//---------------------------------------------------------------------------------------------------------------
//
//  HAUD 2023.03.07
//
//  - XTS_TRANSPORT_LAYER
//
//  fb_Station
//  - handshake with extern control for mover transport through station
//
//---------------------------------------------------------------------------------------------------------------
// This SOFTWARE is provided as an Exemple by THE PROVIDER "as is" and "with all faults." THE PROVIDER makes no 
// representations or warranties of any kind concerning the safety, suitability, lack of viruses, inaccuracies, 
// typographical errors, or other harmful components of this SOFTWARE. There are inherent dangers in the use of 
// any software, and you are solely responsible for determining whether this SOFTWARE is compatible with your 
// equipment and other software installed on your equipment. You are also solely responsible for the protection 
// of your equipment and backup of your data, and THE PROVIDER will not be liable for any damages you may suffer 
// in connection with using, modifying, or distributing this SOFTWARE.
//---------------------------------------------------------------------------------------------------------------
FUNCTION_BLOCK fb_Station IMPLEMENTS I_XtsTransport_Station
VAR
  _nStationId                 : UINT;         // why is Gamora?

  _sState                     : STRING(255);  // additional output for Check()

  _eInitList                  : E_PROGRESS;   // linked list initialization progress

  _eFatalError                : E_STATION_STATE;

  // pointer to all stations
  _stCtrl                     : REFERENCE TO ARRAY[1..MAX_STATION]  OF ST_STATION_CTRL;
  _stState                    : REFERENCE TO ARRAY[1..MAX_STATION]  OF ST_STATION_STATE;

  // local copy of command
  _eCmd,
  _eCmdOld                    : E_STATION_CTRL;

  _ItfStation                 : REFERENCE TO ARRAY[1..MAX_STATION]  OF I_Station_LinkedList;  // access to all stations lists
  _ItfMover                   : REFERENCE TO ARRAY[1..MAX_MOVER]    OF I_XtsTransport_Mover;  // access to mover methods

  // station related data
  _rMoverOffset               : REFERENCE TO ARRAY[1..MAX_STATION]  OF T_NEST_OFFSET;         // static offsets for station
  _stParameter                : REFERENCE TO ARRAY[1..MAX_STATION]  OF ST_STATION_PARAMETER;  // station parameter (where, how fast, how many stops)

  // mover axis ref for info
  _Mover                      : REFERENCE TO ARRAY[1..MAX_MOVER]    OF AXIS_REF;              // read from AXIS_REF

  // linked list result struct
  _stListEnter,
  _stListTarget,
  _stListDelete               : ST_STATION_LIST_RESULT;   // struct with result and ticket data

  _stMoverDataSend,
  _stMoverData                : ST_STATION_MOVER_DATA;    // mover ticket data

  _stInfeed,
  _stOutfeed                  : ST_MOVE_DATA;             // position and dynamic constraints of movement

  // work vars
  _Result                     : E_PROGRESS;
  _eStateProgress             : E_PROGRESS;

  _nNest,
  _nMoverDetected,
  _ix                         : UINT;

  _rModActPosFetch            : LREAL;
  _stMsg                      : ST_Message;
  _eMessageLevel              : E_MessageType;
END_VAR

METHOD PRIVATE Check : BOOL
VAR_INPUT
END_VAR
IF NOT (_nStationId > 0) OR
       (_nStationId > MAX_STATION)
THEN
  _sState                     := 'invalid nStationId';
  RETURN;
END_IF

IF NOT __ISVALIDREF(_stCtrl)
THEN
  _sState                     := '_stCtrl: missing pointer';
  RETURN;
END_IF

IF NOT __ISVALIDREF(_stState)
THEN
  _sState                     := '_stState: missing pointer';
  RETURN;
END_IF

IF NOT __ISVALIDREF(_ItfStation)
THEN
  _sState                     := '_ItfStation: missing interface';
  RETURN;
END_IF

IF NOT __ISVALIDREF(_ItfMover)
THEN
  _sState                     := '_ItfMover: missing interface';
  RETURN;
END_IF

IF NOT __ISVALIDREF(_rMoverOffset)
THEN
  _sState                     := '_rMoverOffset: missing pointer';
  RETURN;
END_IF

IF NOT __ISVALIDREF(_stParameter)
THEN
  _sState                     := '_stParameter: missing pointer';
  RETURN;
END_IF

IF NOT __ISVALIDREF(_Mover)
THEN
  _sState                     := '_Mover: missing pointer';
  RETURN;
END_IF


_sState                       := 'CHECK_DONE';
Check                         := TRUE;
END_METHOD

PROPERTY Ctrl : reference to ARRAY[1..MAX_STATION] OF ST_STATION_CTRL
SET
_stCtrl ref= Ctrl;
END_SET
END_PROPERTY

METHOD Cycle
//-----------------------------------------------------------------------------
//-----------------------------------------------------------------------------
// check pointer and interface
//-----------------------------------------------------------------------------
IF NOT Check() THEN RETURN; END_IF
//-----------------------------------------------------------------------------
//-----------------------------------------------------------------------------
// set message device ID
//-----------------------------------------------------------------------------
_stMsg.eDevice                        := e_Device.XtsStation + _nStationId;
//-----------------------------------------------------------------------------
//-----------------------------------------------------------------------------
// log command change
//-----------------------------------------------------------------------------
_eCmd                                 := _stCtrl[_nStationId].eCmd;
IF (_eCmd <> _eCmdOld)
THEN
  _eCmdOld                            := _eCmd;

  _stMsg.eType                        := E_MessageType.eMessageInfo;
  _stMsg.eSubdevice                   := StationControl;
  _stMsg.iErrorNumber                 := 0;
  _stMsg.sText                        := TO_STRING(_eCmd);

  IF (_eMessageLevel > E_MessageType.eMessageWarning)
  THEN
    f_MessageSet(_stMsg);
  END_IF
END_IF
//-----------------------------------------------------------------------------
//-----------------------------------------------------------------------------
// clear station on demand
//-----------------------------------------------------------------------------
CASE _stCtrl[_nStationId].eCmd
OF
  E_STATION_CTRL.STATION_INIT:        // commanded init from cyclic interface
    _eInitList                        := Init();
    _stState[_nStationId].rMoverModPos:= 0.0;
    _stState[_nStationId].nQueue      := TO_USINT(_ItfStation[_nStationId].Count);
    RETURN;
END_CASE
//-----------------------------------------------------------------------------
//-----------------------------------------------------------------------------
// station startup and init states
//-----------------------------------------------------------------------------
CASE _stState[_nStationId].eState
OF
  E_STATION_STATE.STATION_NO_INIT:    // startup state in first PLC cycle, init linked list required
    _eInitList                        := Init();

  E_STATION_STATE.STATION_INIT:       // switch state as reserve for anything you might add here
    _stState[_nStationId].eState      := E_STATION_STATE.STATION_DISABLE;
END_CASE
//-----------------------------------------------------------------------------
//-----------------------------------------------------------------------------
//  station disabled after init 
//  wait for command to enable
//  return state after a mover has left station
//  fall back state before entry was allowed and you decided to disable
//-----------------------------------------------------------------------------
CASE _stState[_nStationId].eState
OF
  E_STATION_STATE.STATION_DISABLE:
    IF (_stCtrl[_nStationId].eCmd = E_STATION_CTRL.STATION_ENABLE)
    THEN
      _stState[_nStationId].eState    := E_STATION_STATE.STATION_ENABLE;
    END_IF


  E_STATION_STATE.STATION_ENABLE:     // enable state is detectable on the interface for one cycle only
                                      // double check commanded enable and clear work vars
    IF (_stCtrl[_nStationId].eCmd = E_STATION_CTRL.STATION_DISABLE)
    THEN
      _stState[_nStationId].eState    := E_STATION_STATE.STATION_DISABLE;
    ELSE
      memset(ADR(_stListEnter),    0, SIZEOF(_stListEnter));

      _eStateProgress                 := E_PROGRESS.PROGRESS_INIT;  // substate for procedures within one state
      _stState[_nStationId].eState    := E_STATION_STATE.STATION_DETECT_MOVER;  // switch to mover detection

      IF (_eMessageLevel = E_MessageType.eMessageVerbose)
      THEN
        _stMsg.eType                  := _eMessageLevel;
        LogState(_stMsg.eType);
      END_IF
    END_IF
END_CASE
//-----------------------------------------------------------------------------
//-----------------------------------------------------------------------------
//  detection state
//   - wait until mover data is entered into list
//
//  check for disable command; fall back to disabled state
//  check linked list for new entry; proceed to request infeed of mover
//-----------------------------------------------------------------------------
CASE _stState[_nStationId].eState
OF
  E_STATION_STATE.STATION_DETECT_MOVER:// wait state for mover detection
    CASE _eStateProgress
    OF
      E_PROGRESS.PROGRESS_INIT:
        IF (_stCtrl[_nStationId].eCmd = E_STATION_CTRL.STATION_DISABLE) // check for commanded disable
        THEN
          IF (_eMessageLevel = E_MessageType.eMessageVerbose)
          THEN
            _stMsg.eType              := E_MessageType.eMessageVerbose;
            _stMsg.eSubdevice         := Stationstate;
            _stMsg.iErrorNumber       := _stState[_nStationId].nMoverId;
            _stMsg.sText              := concat(TO_STRING(_stState[_nStationId].eState), ': ');
            _stMsg.sText              := concat(_stMsg.sText, TO_STRING(E_STATION_STATE.STATION_DISABLE));
            f_MessageSet(_stMsg);
          END_IF
          _stState[_nStationId].eState      := E_STATION_STATE.STATION_DISABLE; // go back and wait, no matter the queue

        ELSIF (_ItfStation[_nStationId].Count > 0)
        THEN
          // someone entered something in my list
          _stListEnter                := _ItfStation[_nStationId].GetHead();
          _eStateProgress             := E_PROGRESS.PROGRESS_BUSY;  // go check list result data

          IF (_eMessageLevel > E_MessageType.eMessageWarning)
          THEN
            _stMsg.eType              := E_MessageType.eMessageInfo;
            _stMsg.eSubdevice         := Stationstate;
            _stMsg.iErrorNumber       := _stState[_nStationId].nMoverId;
            _stMsg.sText              := concat(TO_STRING(_stState[_nStationId].eState), ': ');
            _stMsg.sText              := concat(_stMsg.sText, TO_STRING(_eStateProgress));
            f_MessageSet(_stMsg);
          END_IF
        END_IF
    END_CASE
    CASE _eStateProgress
    OF
      E_PROGRESS.PROGRESS_BUSY:
        IF (_stListEnter.wState = 0)  // GetHead() without error
        THEN
          _stMsg.eType                := E_MessageType.eMessageVerbose;
          _stMsg.eSubdevice           := e_Subdevice.StationGetHead;
          _stMsg.iErrorNumber         := _stListEnter.stData.nMoverId;
          _stMsg.sText                := '';
          IF (_eMessageLevel = E_MessageType.eMessageVerbose)
          THEN
            f_MessageSet(_stMsg);
          END_IF

          // list is giving head as result
          _stMoverData                := _stListEnter.stData; // copy ticket from list result
          _eStateProgress             := E_PROGRESS.PROGRESS_PREPARE; // go check plausibility of ticket

          IF (_eMessageLevel = E_MessageType.eMessageVerbose)
          THEN
            _stMsg.eType              := E_MessageType.eMessageVerbose;
            _stMsg.eSubdevice         := Stationstate;
            _stMsg.iErrorNumber       := _stState[_nStationId].nMoverId;
            _stMsg.sText              := concat(TO_STRING(_stState[_nStationId].eState), ': ');
            _stMsg.sText              := concat(_stMsg.sText, TO_STRING(_eStateProgress));
            f_MessageSet(_stMsg);
          END_IF
        ELSE
          // the thing that must not be: GetHead() with error
          _stState[_nStationId].eState      := E_STATION_STATE.STATION_ERROR_LIST_GET_HEAD_FAULT; // fatal error

          _stMsg.eType                      := E_MessageType.eMessageError;
          LogState(_stMsg.eType);
        END_IF
    END_CASE
    CASE _eStateProgress
    OF
      E_PROGRESS.PROGRESS_PREPARE:    // check ticket (list entry)
        // check target assignement
        IF NOT (_stMoverData.nTargetStation = _nStationId)
        THEN
          // for whom the mover calls
          // wrong address, right mover?
          _stState[_nStationId].eState      := E_STATION_STATE.STATION_ERROR_LIST_STATION_ID_WRONG; // ctrl has to fix this, go tell ctrl

          _stMsg.eType                      := E_MessageType.eMessageWarning;
          LogState(_stMsg.eType);
        ELSE
          // it's a me
          _nMoverDetected                   := _stMoverData.nMoverId;

          IF (_nMoverDetected < 1) OR
             (_nMoverDetected > MAX_MOVER)
          THEN
            // out of range the mover must not be
            _stState[_nStationId].eState    := E_STATION_STATE.STATION_ERROR_LIST_MOVER_ID_INVALID; // fatal error

            _stMsg.eType                    := E_MessageType.eMessageError;
            LogState(_stMsg.eType);
          ELSE
            memset(ADR(_stListDelete),   0, SIZEOF(_stListDelete)); // clear work var
            _eStateProgress                 := E_PROGRESS.PROGRESS_INIT; // clear progress for next station state

            // prepare station state for new mover
            _stState[_nStationId].nMoverId  := TO_USINT(_nMoverDetected); // who is waiting to enter
            _stState[_nStationId].nMask     := _stMoverData.nMask;        // how many stops have to be made
            _stState[_nStationId].eState    := E_STATION_STATE.STATION_MOVER_ENTER; // go ask for permission to enter

            IF (_eMessageLevel > E_MessageType.eMessageWarning)
            THEN
              _stMsg.eType            := E_MessageType.eMessageInfo;
              _stMsg.eSubdevice       := Stationstate;
              _stMsg.iErrorNumber     := _stState[_nStationId].nMoverId;
              _stMsg.sText            := concat(TO_STRING(_stState[_nStationId].eState), ': ');
              _stMsg.sText            := concat(_stMsg.sText, TO_STRING(_eStateProgress));
              f_MessageSet(_stMsg);
            END_IF
          END_IF
        END_IF
    END_CASE
END_CASE
//-----------------------------------------------------------------------------
//-----------------------------------------------------------------------------
// enter into station state
//  last check for disable command; fall back to disabled state
//  check for command to enter; prepare moverment, start movement
//  check for command to skip; prepare movement, switch to outfeed state
//-----------------------------------------------------------------------------
CASE _stState[_nStationId].eState
OF
  E_STATION_STATE.STATION_MOVER_ENTER:          // requesting permission for mover to enter station
    CASE _eStateProgress
    OF
      E_PROGRESS.PROGRESS_INIT:

        CASE _stCtrl[_nStationId].eCmd
        OF
          E_STATION_CTRL.STATION_DISABLE:       // control decided to disable, mover will wait
            _stState[_nStationId].eState    := E_STATION_STATE.STATION_DISABLE;

            IF (_eMessageLevel = E_MessageType.eMessageVerbose)
            THEN
              _stMsg.eType                  := _eMessageLevel;
              LogState(_stMsg.eType);
            END_IF

          E_STATION_CTRL.STATION_MOVER_ENTER:   // control decided to let mover enter
            _nNest                    := 1;     // default nest/PosStop[1]
            _eStateProgress           := E_PROGRESS.PROGRESS_BUSY;

            IF (_eMessageLevel = E_MessageType.eMessageVerbose)
            THEN
              _stMsg.eType            := E_MessageType.eMessageVerbose;
              _stMsg.eSubdevice       := Stationstate;
              _stMsg.iErrorNumber     := _stState[_nStationId].nMoverId;
              _stMsg.sText            := concat(TO_STRING(_stState[_nStationId].eState), ': ');
              _stMsg.sText            := concat(_stMsg.sText, TO_STRING(_eStateProgress));
              f_MessageSet(_stMsg);
            END_IF

            FOR _ix := 1 TO _stParameter[_nStationId].nConfiguredStopCount
            DO
              IF GetBitWord(_stMoverData.nMask, _ix-1)
              THEN
                _nNest                := _ix;
                EXIT;
              END_IF
            END_FOR

          E_STATION_CTRL.STATION_MOVER_SEND:    // control decided to send mover away
            _stOutfeed.rDistance          := _stParameter[_nStationId].rReleaseDistance;
            _stState[_nStationId].eState  := E_STATION_STATE.STATION_MOVER_OUT;

            IF (_eMessageLevel = E_MessageType.eMessageVerbose)
            THEN
              _stMsg.eType                := _eMessageLevel;
              LogState(_stMsg.eType);
            END_IF
        END_CASE
    END_CASE
    CASE _eStateProgress
    OF
      E_PROGRESS.PROGRESS_BUSY:
        MoveData();                   // prepare movement into station

        // check if infeed movement has to cross modulo turn
        _rModActPosFetch              := _Mover[_stMoverData.nMoverId].NcToPlc.ModuloActPos;

        IF (_rModActPosFetch > _stInfeed.rPos + _stParameter[_nStationId].rReleaseDistance)
        THEN
          _stInfeed.rPos              := _stInfeed.rPos + TO_REAL(_ItfMover[_stMoverData.nMoverId].RailLength);
        END_IF

        _stState[_nStationId].eState  := E_STATION_STATE.STATION_MOVER_IN_TARGET;

        IF (_eMessageLevel = E_MessageType.eMessageVerbose)
        THEN
          _stMsg.eType                := _eMessageLevel;
          LogState(_stMsg.eType);
        END_IF
    END_CASE
END_CASE
//-----------------------------------------------------------------------------
//-----------------------------------------------------------------------------
// move into station state
//  wait for movement to be done; mover in position and standstill
//    switch state to process handshake
//-----------------------------------------------------------------------------
CASE _stState[_nStationId].eState
OF
  E_STATION_STATE.STATION_MOVER_IN_TARGET:
    _ItfMover[_stMoverData.nMoverId].MessageLevel := _eMessageLevel;

    _Result := _ItfMover[_stState[_nStationId].nMoverId].MoveToPosCa(TRUE, _stInfeed);

    IF (_Result = E_PROGRESS.PROGRESS_DONE)
    THEN
      // mother! has arrived
      _ItfMover[_stState[_nStationId].nMoverId].MoveToPosCa(FALSE, _stInfeed);
      _stState[_nStationId].eState    := E_STATION_STATE.STATION_PROCESS_START;

      IF (_eMessageLevel > E_MessageType.eMessageWarning)
      THEN
        _stMsg.eType                  := E_MessageType.eMessageInfo;
        LogState(_stMsg.eType);
      END_IF
    ELSE
      IF (_Result = E_PROGRESS.PROGRESS_ERROR)
      THEN
        _ItfMover[_stState[_nStationId].nMoverId].MoveToPosCa(FALSE, _stInfeed);
        _stState[_nStationId].eState  := E_STATION_STATE.STATION_ERROR_INFEED_ERROR; // ctrl has to fix this, go tell ctrl

        _stMsg.eType                  := E_MessageType.eMessageError;
        LogState(_stMsg.eType);
      END_IF 
    END_IF
END_CASE
//-----------------------------------------------------------------------------
//-----------------------------------------------------------------------------
// process handshake state
//  clear bit in mask
//-----------------------------------------------------------------------------
CASE _stState[_nStationId].eState
OF
  E_STATION_STATE.STATION_PROCESS_START:
    IF (_stCtrl[_nStationId].eCmd = E_STATION_CTRL.STATION_PROCESS_START) OR  // double handshake, your choice
       (_stCtrl[_nStationId].eCmd = E_STATION_CTRL.STATION_PROCESS_DONE)      // single handshake, your choice
    THEN
      // clear bit in mask when started/done
      _stState[_nStationId].nMask     := TO_USINT(DelBitWord(TO_WORD(_stState[_nStationId].nMask), _nNest-1));
      _stState[_nStationId].eState    := E_STATION_STATE.STATION_PROCESS_DONE;

      IF (_eMessageLevel = E_MessageType.eMessageVerbose)
      THEN
        _stMsg.eType                  := _eMessageLevel;
        LogState(_stMsg.eType);
      END_IF
    END_IF
END_CASE
//-----------------------------------------------------------------------------
//-----------------------------------------------------------------------------
CASE _stState[_nStationId].eState
OF
  E_STATION_STATE.STATION_PROCESS_DONE:
    IF (_stCtrl[_nStationId].eCmd = E_STATION_CTRL.STATION_PROCESS_DONE)
    THEN
      _stState[_nStationId].eState    := E_STATION_STATE.STATION_CHECK;
    END_IF
END_CASE
//-----------------------------------------------------------------------------
//-----------------------------------------------------------------------------
// check state if the mover has to move to another nest or must leave station
//-----------------------------------------------------------------------------
CASE _stState[_nStationId].eState
OF
  E_STATION_STATE.STATION_CHECK:
    IF (_stState[_nStationId].nMask = 0)
    THEN
      // mover has to leave
      _stState[_nStationId].eState    := E_STATION_STATE.STATION_MOVER_OUT;

      IF (_eMessageLevel = E_MessageType.eMessageVerbose)
      THEN
        _stMsg.eType                  := _eMessageLevel;
        LogState(_stMsg.eType);
      END_IF
    ELSE
      // _stState[_nStationId].nMask <> 0
      FOR _ix := 1 TO MAX_STATION_NEST
      DO
        IF NOT (_ix > _stParameter[_nStationId].nConfiguredStopCount)
        THEN
          IF GetBitWord(_stState[_nStationId].nMask, _ix-1)
          THEN
            // more work to do
            _stState[_nStationId].eState  := E_STATION_STATE.STATION_CHECK_NEST;
            _nNest                        := _ix; // index to move to

            IF (_eMessageLevel = E_MessageType.eMessageVerbose)
            THEN
              _stMsg.eType                := _eMessageLevel;
              LogState(_stMsg.eType);
            END_IF
            EXIT;
          END_IF
        ELSE
          IF GetBitWord(_stState[_nStationId].nMask, _ix-1)
          THEN
            // not configured, not worked
            _stMsg.eType              := E_MessageType.eMessageWarning;
            _stMsg.eSubdevice         := Stationstate;
            _stMsg.iErrorNumber       := _ix;
            _stMsg.sText              := concat(TO_STRING(_stState[_nStationId].eState), ': ');
            _stMsg.sText              := concat(_stMsg.sText, Tc2_Utilities.BYTE_TO_BINSTR(_stState[_nStationId].nMask, TO_INT(MAX_STATION_NEST)));
            IF (_eMessageLevel > E_MessageType.eMessageError)
            THEN
              f_MessageSet(_stMsg);
            END_IF

            _stState[_nStationId].nMask := TO_USINT(DelBitWord(TO_WORD(_stState[_nStationId].nMask), _ix-1));
          END_IF
        END_IF
      END_FOR
    END_IF
END_CASE
//-----------------------------------------------------------------------------
//-----------------------------------------------------------------------------
// wait state before movement to next nest has to be started
//-----------------------------------------------------------------------------
CASE _stState[_nStationId].eState
OF
  E_STATION_STATE.STATION_CHECK_NEST:
    MoveData();

    IF (_stCtrl[_nStationId].eCmd = E_STATION_CTRL.STATION_MOVER_ENTER)
    THEN
      _stState[_nStationId].eState    := E_STATION_STATE.STATION_MOVER_IN_TARGET;
  
      IF (_eMessageLevel = E_MessageType.eMessageVerbose)
      THEN
        _stMsg.eType                  := _eMessageLevel;
        LogState(_stMsg.eType);
      END_IF
    END_IF
END_CASE
//-----------------------------------------------------------------------------
//-----------------------------------------------------------------------------
// wait state for outfeed of mover
//  check ctrl data, target must be plausible, nTargetStation is what you have to set
//-----------------------------------------------------------------------------
CASE _stState[_nStationId].eState
OF
  E_STATION_STATE.STATION_MOVER_OUT:
    IF (_stCtrl[_nStationId].eCmd = E_STATION_CTRL.STATION_MOVER_OUT)
    THEN
      IF (_stCtrl[_nStationId].nTargetStation < 1) OR  
         (_stCtrl[_nStationId].nTargetStation > MAX_STATION)
      THEN
        _stState[_nStationId].eState  := E_STATION_STATE.STATION_ERROR_OUTFEED_TARGET_INVALID; // ctrl has to fix this, go tell ctrl

        _stMsg.eType                  := E_MessageType.eMessageError;
        LogState(_stMsg.eType);
      ELSE
        _stListDelete                 := _ItfStation[_nStationId].RemoveHeadValue(); // delete mover data in stations linked list


        IF (_stListDelete.wState <> 0)
        THEN
        // deleting mover in list was NOT successful
          _stState[_nStationId].eState:= E_STATION_STATE.STATION_ERROR_LIST_REMOVE_HEAD_FAULT; // fatal error

          _stMsg.eType                := E_MessageType.eMessageError;
          LogState(_stMsg.eType);

        ELSE
        // mover data successfully deleted
          _stMsg.eType                := E_MessageType.eMessageVerbose;
          _stMsg.eSubdevice           := e_Subdevice.StationRemoveHeadValue;
          _stMsg.iErrorNumber         := _stState[_nStationId].nMoverId;
          _stMsg.sText                := '';
          IF (_eMessageLevel = E_MessageType.eMessageVerbose)
          THEN
            f_MessageSet(_stMsg);
          END_IF

          memset(ADR(_stListTarget),   0, SIZEOF(_stListTarget)); // clear debug var

          // prepare movement and switch state to start movement
          MoverOut();
          _stState[_nStationId].eState  := E_STATION_STATE.STATION_MOVER_RELEASE;

          IF (_eMessageLevel > E_MessageType.eMessageWarning)
          THEN
            _stMsg.eType                := E_MessageType.eMessageInfo;
            LogState(_stMsg.eType);
          END_IF
        END_IF
      END_IF
    END_IF
END_CASE
//-----------------------------------------------------------------------------
//-----------------------------------------------------------------------------
// ckeck if mover has left the station
//  enter mover data into list of target station
//-----------------------------------------------------------------------------
CASE _stState[_nStationId].eState
OF
  E_STATION_STATE.STATION_MOVER_RELEASE:
    _ItfMover[_stMoverData.nMoverId].MessageLevel := _eMessageLevel;

    _Result                           := _ItfMover[_stMoverDataSend.nMoverId].SendToModuloPosCa(TRUE, _stOutfeed);

    IF (_Result = E_PROGRESS.PROGRESS_DONE)
    THEN
      // add entry in target station list
      _stListTarget                   := _ItfStation[_stMoverDataSend.nTargetStation].AddTailValue(_stMoverDataSend);

      IF (_stListTarget.wState <> 0)
      THEN
      // adding mover in target list was NOT successful
        _stState[_nStationId].eState  := E_STATION_STATE.STATION_ERROR_LIST_ADD_TAIL_FAULT; // fatal error
        _stMsg.eType                  := E_MessageType.eMessageError;
        LogState(_stMsg.eType);

      ELSE
      // mover data successfully added to target station list
        IF (_eMessageLevel > E_MessageType.eMessageWarning)
        THEN
          _stMsg.eType                := E_MessageType.eMessageInfo;
          _stMsg.eSubdevice           := e_Subdevice.StationAddTail;
          _stMsg.iErrorNumber         := _stState[_nStationId].nMoverId;
          _stMsg.sText                := concat('TargetStation: ', TO_STRING(_stListTarget.stData.nTargetStation));
          f_MessageSet(_stMsg);
        END_IF

        _stState[_nStationId].eState  := E_STATION_STATE.STATION_MOVER_GONE; // go tell ctrl that station is empty

        IF (_eMessageLevel = E_MessageType.eMessageVerbose)
        THEN
          _stMsg.eType                := _eMessageLevel;
          LogState(_stMsg.eType);
        END_IF
      END_IF
    ELSIF (_Result = E_PROGRESS.PROGRESS_ERROR)
    THEN
      _stState[_nStationId].eState    := E_STATION_STATE.STATION_ERROR_OUTFEED_ERROR; // ctrl has to fix this, go tell ctrl
      _stMsg.eType                    := E_MessageType.eMessageError;
      LogState(_stMsg.eType);
    END_IF
END_CASE
//-----------------------------------------------------------------------------
//-----------------------------------------------------------------------------
// check handshake for empty station
//  switch back station state for new mover to be able to enter
//-----------------------------------------------------------------------------
CASE _stState[_nStationId].eState
OF
  E_STATION_STATE.STATION_MOVER_GONE:
    _ItfMover[_stMoverDataSend.nMoverId].SendToModuloPosCa(FALSE, _stOutfeed);

    memset(ADR(_stMoverData),  0, SIZEOF(_stMoverData));

    _stState[_nStationId].nMask       := 0;
    _stState[_nStationId].nMoverId    := 0;

    IF (_stCtrl[_nStationId].eCmd = E_STATION_CTRL.STATION_MOVER_GONE)
    THEN
      _stState[_nStationId].eState    := E_STATION_STATE.STATION_DISABLE;

      IF (_eMessageLevel = E_MessageType.eMessageVerbose)
      THEN
        _stMsg.eType                  := _eMessageLevel;
        LogState(_stMsg.eType);
      END_IF
    END_IF
END_CASE
//-----------------------------------------------------------------------------
//-----------------------------------------------------------------------------
_sState                               := TO_STRING(_stState[_nStationId].eState);
//-----------------------------------------------------------------------------
//-----------------------------------------------------------------------------
// Error handling
//-----------------------------------------------------------------------------
CASE _stState[_nStationId].eState
OF
  //---------------------------------------------------------------------------
  //---------------------------------------------------------------------------
  E_STATION_STATE.STATION_ERROR_LIST_STATION_ID_WRONG:
    IF (_stCtrl[_nStationId].eCmd = E_STATION_CTRL.STATION_MOVER_OUT)
    THEN
      _nMoverDetected                 := _stMoverData.nMoverId;

      IF (_nMoverDetected < 1) OR
         (_nMoverDetected > MAX_MOVER)
      THEN
        // this MUST NOT happen
        _stState[_nStationId].eState  := E_STATION_STATE.STATION_ERROR_LIST_MOVER_ID_INVALID; // fatal error
        _stMsg.eType                  := E_MessageType.eMessageError;
        LogState(_stMsg.eType);

      ELSE
        // not for station; send mover out
        _stState[_nStationId].eState  := E_STATION_STATE.STATION_MOVER_OUT;

        IF (_eMessageLevel > E_MessageType.eMessageError)
        THEN
          _stMsg.eType                := E_MessageType.eMessageInfo;
          LogState(_stMsg.eType);
        END_IF
      END_IF

    ELSIF (_stCtrl[_nStationId].eCmd = E_STATION_CTRL.STATION_MOVER_ENTER)
    THEN
      // override wrong TargetStationId in List; start infeed of mover

      _nMoverDetected                 := _stMoverData.nMoverId;

      IF (_nMoverDetected < 1) OR
         (_nMoverDetected > MAX_MOVER)
      THEN
        // this MUST NOT happen
        _stState[_nStationId].eState  := E_STATION_STATE.STATION_ERROR_LIST_MOVER_ID_INVALID; // fatal error

        _stMsg.eType                  := E_MessageType.eMessageError;
        LogState(_stMsg.eType);

      ELSE
        _eStateProgress               := E_PROGRESS.PROGRESS_INIT;
        _stState[_nStationId].nMoverId:= TO_USINT(_nMoverDetected);
        _stState[_nStationId].nMask   := _stMoverData.nMask;
        _stState[_nStationId].eState  := E_STATION_STATE.STATION_MOVER_ENTER;

        IF (_eMessageLevel > E_MessageType.eMessageError)
        THEN
          _stMsg.eType                := E_MessageType.eMessageInfo;
          LogState(_stMsg.eType);
        END_IF
      END_IF
    END_IF

  //---------------------------------------------------------------------------
  //---------------------------------------------------------------------------
  E_STATION_STATE.STATION_ERROR_OUTFEED_TARGET_INVALID:
    // wait here until valid target is detected
    IF NOT (_stCtrl[_nStationId].nTargetStation < 1) AND  
       NOT (_stCtrl[_nStationId].nTargetStation > MAX_STATION)
    THEN
      _stState[_nStationId].eState    := E_STATION_STATE.STATION_MOVER_OUT;

      IF (_eMessageLevel > E_MessageType.eMessageError)
      THEN
        _stMsg.eType                  := E_MessageType.eMessageInfo;
        LogState(_stMsg.eType);
      END_IF
    END_IF

  //---------------------------------------------------------------------------
  //---------------------------------------------------------------------------
  E_STATION_STATE.STATION_ERROR_INFEED_ERROR:   // must be fixed by extern by using cyclic mover control
    IF (_stCtrl[_nStationId].eCmd = E_STATION_CTRL.STATION_MOVER_ENTER_RETRY)
    THEN
      _stState[_nStationId].eState    := E_STATION_STATE.STATION_DETECT_MOVER;   // return to start and wait

      IF (_eMessageLevel > E_MessageType.eMessageError)
      THEN
        _stMsg.eType                  := E_MessageType.eMessageInfo;
        LogState(_stMsg.eType);
      END_IF
    END_IF


  //---------------------------------------------------------------------------
  //---------------------------------------------------------------------------
  E_STATION_STATE.STATION_ERROR_OUTFEED_ERROR:  // must be fixed by extern by using cyclic mover control
    IF (_stCtrl[_nStationId].eCmd = E_STATION_CTRL.STATION_MOVER_OUT_RETRY)
    THEN
      _stState[_nStationId].eState    := E_STATION_STATE.STATION_MOVER_OUT; // return to send out and wait

      IF (_eMessageLevel > E_MessageType.eMessageError)
      THEN
        _stMsg.eType                  := E_MessageType.eMessageInfo;
        LogState(_stMsg.eType);
      END_IF

    ELSIF (_stCtrl[_nStationId].eCmd = E_STATION_CTRL.STATION_MOVER_GONE)
    THEN
      MoverOut();

      // add entry in target station list
      _stListTarget                   := _ItfStation[_stMoverDataSend.nTargetStation].AddTailValue(_stMoverDataSend);
      IF (_stListTarget.wState <> 0)
      THEN
        _stState[_nStationId].eState  := E_STATION_STATE.STATION_ERROR_LIST_ADD_TAIL_FAULT; // fatal error
        _stMsg.eType                  := E_MessageType.eMessageError;
        LogState(_stMsg.eType);

      ELSE
        IF (_eMessageLevel > E_MessageType.eMessageError)
        THEN
          _stMsg.eType                := E_MessageType.eMessageInfo;
          _stMsg.eSubdevice           := e_Subdevice.StationAddTail;
          _stMsg.iErrorNumber         := _stState[_nStationId].nMoverId;
          _stMsg.sText                := concat('TargetStation: ', TO_STRING(_stListTarget.stData.nTargetStation));
          f_MessageSet(_stMsg);
        END_IF

        _stState[_nStationId].eState  := E_STATION_STATE.STATION_MOVER_GONE;

        IF (_eMessageLevel > E_MessageType.eMessageError)
        THEN
          _stMsg.eType                := E_MessageType.eMessageInfo;
          LogState(_stMsg.eType);
        END_IF
      END_IF
    END_IF

  //---------------------------------------------------------------------------
  // fatal errors
  //---------------------------------------------------------------------------
  E_STATION_STATE.STATION_ERROR_LIST_GET_HEAD_FAULT,
  E_STATION_STATE.STATION_ERROR_LIST_REMOVE_HEAD_FAULT,
  E_STATION_STATE.STATION_ERROR_LIST_ADD_TAIL_FAULT,
  E_STATION_STATE.STATION_ERROR_LIST_MOVER_ID_INVALID:
    _stMsg.eType                      := E_MessageType.eMessageError;
    LogState(_stMsg.eType);
    // yes, but why?
    // cannot be fixed by ctrl
    _eFatalError                      := _stState[_nStationId].eState;
    _stState[_nStationId].eState      := E_STATION_STATE.STATION_ERROR_FATAL;
    LogState(_stMsg.eType);

  //---------------------------------------------------------------------------
  //---------------------------------------------------------------------------
  E_STATION_STATE.STATION_ERROR_FATAL:
    // write to string for debugging
    _sState                           := concat(TO_STRING(_stState[_nStationId].eState), ': ');
    _sState                           := concat(_sState, TO_STRING(_eFatalError));
END_CASE
//-----------------------------------------------------------------------------
//-----------------------------------------------------------------------------
IF (_stState[_nStationId].nMoverId > 0) AND
   (_stState[_nStationId].nMoverId < MAX_MOVER+1)
THEN
  _stState[_nStationId].rMoverModPos  := _Mover[_stState[_nStationId].nMoverId].NcToPlc.ModuloActPos;
END_IF
//-----------------------------------------------------------------------------
//-----------------------------------------------------------------------------
_stState[_nStationId].nQueue          := TO_USINT(_ItfStation[_nStationId].Count);
//-----------------------------------------------------------------------------
//-----------------------------------------------------------------------------
END_METHOD

METHOD PUBLIC DelBitWord : WORD
VAR_INPUT
  inVal   : WORD;
  bitNo   : DINT;
END_VAR
VAR
  wConst : WORD := 1;
END_VAR
IF ( inVal AND SHL( wConst, TO_SINT(bitNo) MOD 16 ) ) > 0 THEN
  DelBitWord := inVal XOR (SHL( wConst,TO_SINT(bitNo) MOD 16 ));
ELSE
  DelBitWord := inVal;
END_IF
END_METHOD

METHOD PUBLIC GetBitWord : BOOL
VAR_INPUT
  inVal   : WORD;
  bitNo   : DINT;
END_VAR
VAR
  wConst : WORD := 1;
END_VAR
IF ( inVal AND SHL( wConst,TO_SINT(bitNo) MOD 16 ) ) > 0
THEN
  GetBitWord := TRUE;
ELSE
  GetBitWord := FALSE;
END_IF
END_METHOD

METHOD Init : e_progress
VAR_INPUT
END_VAR
// check pointer and interface
IF NOT Check() THEN Init := e_progress.PROGRESS_ERROR; RETURN; END_IF

_stState[_nStationId].nMask       := 0;
_stState[_nStationId].nMoverId    := 0;

_eFatalError                      := E_STATION_STATE.STATION_ERROR_NULL;

_stState[_nStationId].eState      := E_STATION_STATE.STATION_INIT;
_sState                           := TO_STRING(_stState[_nStationId].eState);

IF _ItfStation[_nStationId].InitList()
THEN
  IF (_eMessageLevel = E_MessageType.eMessageVerbose)
  THEN
    _stMsg.eType                  := E_MessageType.eMessageVerbose;
    _stMsg.eSubdevice             := Stationstate;
    _stMsg.iErrorNumber           := 0;
    _stMsg.sText                  := concat('_ItfStation.InitList', ': ');
    _stMsg.sText                  := concat(_stMsg.sText, TO_STRING(E_PROGRESS.PROGRESS_DONE));
    //f_MessageSet(_stMsg);
  END_IF

  Init                            := E_PROGRESS.PROGRESS_DONE;

ELSE
    _stMsg.eType                  := E_MessageType.eMessageError;
    _stMsg.eSubdevice             := Stationstate;
    _stMsg.iErrorNumber           := 0;
    _stMsg.sText                  := concat('_ItfStation.InitList', ': ');
    _stMsg.sText                  := concat(_stMsg.sText, TO_STRING(E_PROGRESS.PROGRESS_ERROR));
    f_MessageSet(_stMsg);

  Init                            := e_progress.PROGRESS_ERROR;
END_IF
END_METHOD

PROPERTY ItfMover : reference to ARRAY[1..MAX_MOVER] OF I_XtsTransport_Mover
SET
_ItfMover ref= ItfMover;
END_SET
END_PROPERTY

PROPERTY ItfStations : reference to ARRAY[1..MAX_STATION] OF I_Station_LinkedList
SET
_ItfStation ref= ItfStations;
END_SET
END_PROPERTY

METHOD LogState
VAR_INPUT
  eType       : E_MessageType;
END_VAR
_stMsg.eType                := eType;
_stMsg.eSubdevice           := Stationstate;
_stMsg.iErrorNumber         := _stState[_nStationId].nMoverId;
_stMsg.sText                := TO_STRING(_stState[_nStationId].eState);
f_MessageSet(_stMsg);
END_METHOD

PROPERTY MessageLevel : e_messagetype
SET
_eMessageLevel := MessageLevel;
END_SET
END_PROPERTY

METHOD PRIVATE MoveData // prepares movement to PostStop[_nNest] in station
// build WorkPos from parameter, static station data and information on mover
_stInfeed.rPos            := _stParameter[_nStationId].rPosWait
                          +  _stParameter[_nStationId].rPosStop[_nNest]
                          +  _stMoverData.rOffset
                          +  _rMoverOffset[_nStationId][_stMoverData.nMoverId][_nNest];

_stInfeed.rVelo           := _stParameter[_nStationId].rVelo;
_stInfeed.rAcc            := _stParameter[_nStationId].rAccDec;
_stInfeed.rJerk           := _stParameter[_nStationId].rJerk;
_stInfeed.rGap            := _stParameter[_nStationId].rGap;
_stInfeed.rDistance       := _stParameter[_nStationId].rReleaseDistance;

// init method
_ItfMover[_stState[_nStationId].nMoverId].MoveToPosCa(FALSE, _stInfeed);

// clear substate
_eStateProgress           := E_PROGRESS.PROGRESS_INIT;
END_METHOD

PROPERTY Mover : reference TO ARRAY[1..MAX_MOVER] OF AXIS_REF;
SET
_Mover ref= Mover;
END_SET
END_PROPERTY

PROPERTY MoverOffset : reference TO ARRAY[1..MAX_STATION]  OF T_NEST_OFFSET
SET
_rMoverOffset ref= MoverOffset;
END_SET
END_PROPERTY

METHOD PRIVATE MoverOut // prepares mover data for sending to target station
// build data for sending mover to target station

// who am I sending?
_stMoverDataSend.nMoverId         := _stState[_nStationId].nMoverId;

// get optional information about nests to work
_stMoverDataSend.nMask            := _stCtrl[_nStationId].nMask;

// get optional offset
_stMoverDataSend.rOffset          := _stCtrl[_nStationId].rOffset;

// get target station
_stMoverDataSend.nTargetStation   := _stCtrl[_nStationId].nTargetStation;

// get position of target
_stOutfeed.rPos                   := _stParameter[_stMoverDataSend.nTargetStation].rPosWait;

IF (_stOutfeed.rPos - _Mover[_stMoverDataSend.nMoverId].NcToPlc.ModuloActPos < 0)
THEN
  // only forward, never back
  _stOutfeed.rPos             := _stOutfeed.rPos 
                              +  _ItfMover[_stMoverDataSend.nMoverId].RailLength;
END_IF

_stOutfeed.rVelo              := _stParameter[_nStationId].rVelo;
_stOutfeed.rAcc               := _stParameter[_nStationId].rAccDec;
_stOutfeed.rJerk              := _stParameter[_nStationId].rJerk;
_stOutfeed.rGap               := _stParameter[_nStationId].rGap;
_stOutfeed.rDistance          := _stParameter[_nStationId].rReleaseDistance;

// init method for sending
_ItfMover[_stMoverDataSend.nMoverId].SendToModuloPosCa(FALSE, _stOutfeed);
END_METHOD

METHOD PUBLIC SetBitWord : WORD
VAR_INPUT
  inVal   : WORD;
  bitNo   : DINT;
END_VAR
VAR
  wConst  : WORD := 1;
END_VAR
SetBitWord := inVal OR SHL( wConst,TO_SINT(bitNo) MOD 16 );
END_METHOD

PROPERTY State : reference to ARRAY[1..MAX_STATION] OF ST_STATION_STATE
SET
_stState ref= State;
END_SET
END_PROPERTY

PROPERTY StationId : uint
GET
StationId := _nStationId;
END_GET
SET
_nStationId := StationId;
END_SET
END_PROPERTY

PROPERTY StationParameter : reference TO ARRAY[1..MAX_STATION]  OF ST_STATION_PARAMETER
SET
_stParameter ref= StationParameter;
END_SET
END_PROPERTY

PROPERTY TargetWindow : lreal
GET
TargetWindow := _stInfeed.rDelta;
END_GET
SET
_stInfeed.rDelta := TargetWindow;
END_SET
END_PROPERTY

END_FUNCTION_BLOCK

(* stored: Version 1.1.0.1, ProductVersion 3.1.4024.15
   POU fb_Station: Id {6a0a6a2b-7760-4443-be11-40a67a6801c3}, SpecialFunc None
   Folder methods: Id {ce408873-d67b-4e84-aa34-fd09aafb4812}
   Folder private: Id {479c85c2-0b13-40e4-a114-57671c8eb461}
   Folder properties: Id {1f3172cc-37c1-4ea3-b853-223c95c975ef}
   Method Check: Id {4b557f41-a9d0-445b-87f4-484ea064a02b}
   Property Ctrl: Id {c7c7a006-9961-4a51-a682-221fbb0e325a}
   Set Set: Id {ae2c9079-b5c1-483d-9ce6-0ec6d2b84e7d}
   Method Cycle: Id {7ea7a6f9-8509-4d41-9999-ae04f3572e36}
   Method DelBitWord: Id {1fcb93df-4d80-4b1c-bad6-325007b39b6e}
   Method GetBitWord: Id {3e49b02a-330b-4ba9-b486-d6577a561798}
   Method Init: Id {7504aeb6-1bc5-43b8-9afb-f879fd258e13}
   Property ItfMover: Id {7bb6a22a-6b51-4f72-b870-521d89f00f33}
   Set Set: Id {0b4b65cd-b390-48a7-93c4-92b75e304139}
   Property ItfStations: Id {517c066b-12bc-4649-ad28-04f745e3e87b}
   Set Set: Id {1b66718b-bfc2-427a-b5bd-16809a307b8f}
   Method LogState: Id {8a2a3506-fb04-46f7-8f4b-c3425c424792}
   Property MessageLevel: Id {e61ed6fb-e88b-412a-8b24-37be883dbef9}
   Set Set: Id {2128a689-e668-4b3c-89ed-3ca5af2a1f04}
   Method MoveData: Id {a5a3f59a-6fee-4e82-931e-bcc1715aa98a}
   Property Mover: Id {71ad3ce4-cbc7-4639-ac92-82115d956e55}
   Set Set: Id {f88c8007-8cc1-4951-a2f7-89cddb774ec8}
   Property MoverOffset: Id {b741cb64-939b-4b6a-aa5c-c2510bec8ffb}
   Set Set: Id {22dc33d0-9fef-4026-b28a-3a80ddee0d52}
   Method MoverOut: Id {c53911f4-501b-436e-be79-a75f576784da}
   Method SetBitWord: Id {3f525fda-eedc-431f-9650-e9f04579f12e}
   Property State: Id {915c6493-f92b-4f69-aea4-8517cb57405e}
   Set Set: Id {71d65301-3f8c-45b3-b6ba-502ba104c321}
   Property StationId: Id {2913fa7a-3349-4140-924c-e764850d6b65}
   Get Get: Id {82ac0669-5259-4d6e-84b4-c00fa7dfbed8}
   Set Set: Id {2b36c5d1-50f0-4e81-8e9b-79e222ffdbd0}
   Property StationParameter: Id {4966de79-fe25-4ef3-b797-e0298595abf0}
   Set Set: Id {fabea73f-f7c8-4007-9566-b6f06460640c}
   Property TargetWindow: Id {9ae7cba8-edef-426c-ac3f-c7dae2868a82}
   Get Get: Id {e262fd70-7746-4d93-82ff-17a90d88c3d6}
   Set Set: Id {ddf14a8a-5cc3-4367-927e-abe81cbf72ca} *)
